// TIA Portal V21 export
FUNCTION_BLOCK "Primer_Demo_FB"   // FB120, LAD
TITLE = Primer presentation fixture · 样式示例
// Synthetic offline fixture: contacts, timer, code, an empty network and an existing constant-contact finding. No native export provenance.
   VAR_INPUT
      Enable : Bool := false;
      RampTime : Time := T#2s;
   END_VAR
   VAR_OUTPUT
      Run : Bool;
      RampDone : Bool;
   END_VAR
BEGIN

REGION Network 1: Enable and fault interlock
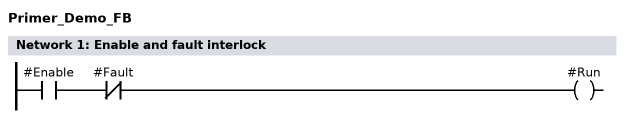
   RUNG wire#powerrail
      Contact( #Enable )
      I_Contact( #Fault )
      Coil( #Run )
   END_RUNG
   // the same network as SCL:
   #Run := #Enable AND NOT #Fault;
END_REGION

REGION Network 2 (FBD): Ramp timer
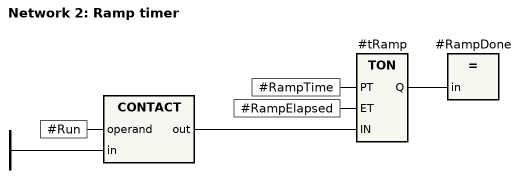
   #tRamp.TON(PT := #RampTime, ET := #RampElapsed, IN := #Run);
   #RampDone := #tRamp.Q;
END_REGION

REGION Network 3 (SCL): Speed limit
   #Speed_SP := LIMIT(MN := 0, IN := #Speed_SP, MX := 100);
END_REGION

REGION Network 5: Constant-contact inspection
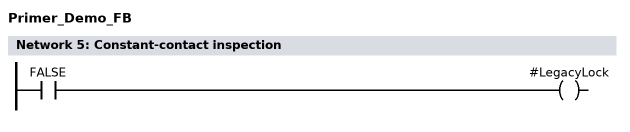
   RUNG wire#powerrail
      Contact( FALSE )
      Coil( #LegacyLock )
   END_RUNG
   // the same network as SCL:
   #LegacyLock := FALSE;
END_REGION
END_FUNCTION_BLOCK
